{attribute addProperty BoxType "EL1502-0000-0018"}
{attribute addProperty Id "CNT_InputsAT %I*CNT_Inputs_917F444B4860CNT_OutputsAT %Q*CNT_Outputs_0B1B8EFA4860WcStateAT %I*WcState_F855686C1620InfoDataAT %I*InfoData_BC63D37F80100"}
{attribute addProperty CRC "610779000"}
{attribute addProperty SizeInBites "192"}
{attribute addProperty SizeInBytes "24"}
TYPE EL1502_C84D344A :
STRUCT
	{attribute addProperty Name "CNT_Inputs"}
	CNT_Inputs : CNT_Inputs_917F444B;
	{attribute addProperty Name "CNT_Outputs"}
	CNT_Outputs : CNT_Outputs_0B1B8EFA;
	{attribute addProperty Name "WcState"}
	WcState : WcState_F855686C;
	{attribute addProperty Name "InfoData"}
	InfoData : InfoData_BC63D37F;
END_STRUCT
END_TYPE

(* stored: Version 1.2.0.0, ProductVersion 3.1.4024.9
   DUT EL1502_C84D344A: Id {441c2563-a45e-442b-87c0-400098cf3428} *)
